{attribute 'qualified_only'}
{attribute 'strict'}
TYPE E_Button :
(
	Start,
	Stop
);
END_TYPE

(* stored: Version 1.1.0.1, ProductVersion 3.1.4024.12
   DUT E_Button: Id {decfa77a-83d1-43f9-893e-3653fce37733} *)
